{attribute addProperty BoxType "IODEVICETYPE_ETHERCATPROT"}
{attribute addProperty Id "Beckhoff_EP1xxxBeckhoff_EP1xxx_C8E7C95B1214068719478253.5Beckhoff_EP2xxxBeckhoff_EP2xxx_B2F46B5A25538171798695032.25Beckhoff_EP3xxxBeckhoff_EP3xxx_2B029919173102163.75Beckhoff_EP4xxxBeckhoff_EP4xxx_3DB4D53F1920240Beckhoff_EP5xxxBeckhoff_EP5xxx_8FA7D6701928241Beckhoff_EP6xxxBeckhoff_EP6xxx_66B3A0F3108981362.25Beckhoff_EP7xxxBeckhoff_EP7xxx_5B32BB7C142491781.125Beckhoff_EP8xxxBeckhoff_EP8xxx_A1F98A041592199Beckhoff_EP9xxxBeckhoff_EP9xxx_40638FD64838604.75SyncUnitsSyncUnits_0037765A39048.75InputsInputs_C75D3FEC1280160OutputsOutputs_47D1E803848106InfoDataInfoData_E9F65A829612"}
{attribute addProperty CRC "2908896672"}
{attribute addProperty SizeInBites "93027"}
{attribute addProperty SizeInBytes "240518180204.375"}
TYPE EtherCAT_Master_EPxxxx_AD623DA0 :
STRUCT
	{attribute addProperty Name "Beckhoff_EP1xxx"}
	Beckhoff_EP1xxx : Beckhoff_EP1xxx_C8E7C95B;
	{attribute addProperty Name "Beckhoff_EP2xxx"}
	Beckhoff_EP2xxx : Beckhoff_EP2xxx_B2F46B5A;
	{attribute addProperty Name "Beckhoff_EP3xxx"}
	Beckhoff_EP3xxx : Beckhoff_EP3xxx_2B029919;
	{attribute addProperty Name "Beckhoff_EP4xxx"}
	Beckhoff_EP4xxx : Beckhoff_EP4xxx_3DB4D53F;
	{attribute addProperty Name "Beckhoff_EP5xxx"}
	Beckhoff_EP5xxx : Beckhoff_EP5xxx_8FA7D670;
	{attribute addProperty Name "Beckhoff_EP6xxx"}
	Beckhoff_EP6xxx : Beckhoff_EP6xxx_66B3A0F3;
	{attribute addProperty Name "Beckhoff_EP7xxx"}
	Beckhoff_EP7xxx : Beckhoff_EP7xxx_5B32BB7C;
	{attribute addProperty Name "Beckhoff_EP8xxx"}
	Beckhoff_EP8xxx : Beckhoff_EP8xxx_A1F98A04;
	{attribute addProperty Name "Beckhoff_EP9xxx"}
	Beckhoff_EP9xxx : Beckhoff_EP9xxx_40638FD6;
	{attribute addProperty Name "SyncUnits"}
	SyncUnits : SyncUnits_0037765A;
	{attribute addProperty Name "Inputs"}
	Inputs : Inputs_C75D3FEC;
	{attribute addProperty Name "Outputs"}
	Outputs : Outputs_47D1E803;
	{attribute addProperty Name "InfoData"}
	InfoData : InfoData_E9F65A82;
END_STRUCT
END_TYPE

(* stored: Version 1.2.0.0, ProductVersion 3.1.4024.9
   DUT EtherCAT_Master_EPxxxx_AD623DA0: Id {c49c9934-6f12-4033-a9c6-1e4a650cd88b} *)
